PROGRAM PRG_TempControl
VAR
	SetPoint			: LREAL := 100;
	ActualTemp	AT %I*	: LREAL;
	Output		AT %Q*	: LREAL;
	fbPID				: FB_CTRL_PID;
	PID_Params			: ST_CTRL_PID_PARAMS := (tCtrlCycleTime	:= TIME#10ms,
												tTaskCycleTime	:= TIME#10ms,
												fKp				:= 10,
												tTn				:= TIME#100ms,
												tTv				:= TIME#45ms,
												tTd				:= TIME#1ms);
END_VAR

fbPID(fSetpointValue := SetPoint,
	fActualValue	:= ActualTemp,
	eMode			:= E_CTRL_MODE.eCTRL_MODE_ACTIVE,
	fOut			=> Output,
	stParams		:= PID_Params);

END_PROGRAM

(* stored: Version 1.1.0.1, ProductVersion 3.1.4024.12
   POU PRG_TempControl: Id {fb6a3f93-c616-41e5-96be-a48c24902e1e}, SpecialFunc None *)
